FUNCTION "GestStazione_PrioritaSerbatoioPerHMI" : Void
{ S7_Optimized_Access := 'TRUE' }
VERSION : 0.1
   VAR_TEMP
      StazioniConPriorità : Array[0.."K_NumStazione"] of Int;
      StazioniSorgenti : Array[0.."K_NumStazione"] of Int;
      StazioniDestinazioni : Array[0.."K_NumStazione"] of Int;
      CounterStazione : Int;
      OccupazioneArray : Int;
      StazioneDaElenco : Int;
      StazioneVisualizzataHmi : Int;
      LeggiDaPlc : Bool;
      LeggiDaHmi : Bool;
   END_VAR


BEGIN
	REGION Pulizia delle temporanee
	    FOR #CounterStazione := 0 TO "K_NumStazione" DO
	        #StazioniSorgenti[#CounterStazione] :=
	        #StazioniDestinazioni[#CounterStazione] :=
	        #StazioniConPriorità[#CounterStazione] := 0;
	    END_FOR;
	    #StazioneVisualizzataHmi := "PrioritaStazioni".K_StazioneVisualizzata;
	END_REGION ;
	REGION Ricerca stazioni con le priorità
	    #OccupazioneArray := 0;
	    FOR #CounterStazione := 0 TO "K_NumStazione" DO
	        IF "Stazione".S[#CounterStazione].Prm.AbilitazionePriorità.SuEstrazioni OR "Stazione".S[#CounterStazione].Prm.AbilitazionePriorità.SugliArrivi THEN
	            #StazioniConPriorità[#OccupazioneArray] := #CounterStazione;
	            #OccupazioneArray += 1;
	        END_IF;
	    END_FOR;
	END_REGION ;
	REGION Ricerca sorgenti e destinazioni per la stazione visualizzata
	    #OccupazioneArray := 0;
	    FOR #CounterStazione := 0 TO "K_NumStazione" DO
	        IF "Stazione".S[#CounterStazione].Destinazione[#StazioneVisualizzataHmi].IN.Possibile THEN
	            #StazioniSorgenti[#OccupazioneArray] := #CounterStazione;
	            #OccupazioneArray += 1;
	        END_IF;
	    END_FOR;
	    #OccupazioneArray := 0;
	    FOR #CounterStazione := 0 TO "K_NumStazione" DO
	        IF "Stazione".S[#StazioneVisualizzataHmi].Destinazione[#CounterStazione].IN.Possibile THEN
	            #StazioniDestinazioni[#OccupazioneArray] := #CounterStazione;
	            #OccupazioneArray += 1;
	        END_IF;
	    END_FOR;
	END_REGION ;
	REGION Definzione dell'elenco di stazioni da visualizzare ad HMI
	    "PrioritaStazioni".K_StazioniSorgenti := #StazioniSorgenti;
	    "PrioritaStazioni".K_StazioniDestinazioni := #StazioniDestinazioni;
	    "PrioritaStazioni".K_StazioniConPriorità := #StazioniConPriorità;
	END_REGION ;
	REGION Definzione lettura e scrittura
	    #LeggiDaPlc := "PrioritaStazioni".Old_K_StazioneVisualizzata <> "PrioritaStazioni".K_StazioneVisualizzata;

	    #LeggiDaHmi :=  ("PrioritaStazioni".Old_StazioniSorgenti_PrioritàHmi <> "PrioritaStazioni".StazioniSorgenti_PrioritàHmi) OR
	                    ("PrioritaStazioni".Old_StazioniDestinazioni_PrioritàHmi <> "PrioritaStazioni".StazioniDestinazioni_PrioritàHmi);
	    IF #LeggiDaPlc THEN
	        FOR #CounterStazione := 0 TO "K_NumStazione" DO
	            #StazioneDaElenco := #StazioniSorgenti[#CounterStazione];    //Sfoglio l'elenco di stazioni e mi salvo la k
	            "PrioritaStazioni".StazioniSorgenti_PrioritàHmi[#CounterStazione] := "Stazione".S[#StazioneDaElenco].Destinazione[#StazioneVisualizzataHmi].Prm.PrioritaRicezioneProdotto;
	        END_FOR;
	        FOR #CounterStazione := 0 TO "K_NumStazione" DO
	            #StazioneDaElenco := #StazioniDestinazioni[#CounterStazione];    //Sfoglio l'elenco di stazioni e mi salvo la k
	            "PrioritaStazioni".StazioniDestinazioni_PrioritàHmi[#CounterStazione] := "Stazione".S[#StazioneVisualizzataHmi].Destinazione[#StazioneDaElenco].Prm.PrioritaInvioProdotto;
	        END_FOR;
	    END_IF;
	    IF #LeggiDaHmi THEN
	        FOR #CounterStazione := 0 TO "K_NumStazione" DO
	            #StazioneDaElenco := #StazioniSorgenti[#CounterStazione];    //Sfoglio l'elenco di stazioni e mi salvo la k
	            "Stazione".S[#StazioneDaElenco].Destinazione[#StazioneVisualizzataHmi].Prm.PrioritaRicezioneProdotto := "PrioritaStazioni".StazioniSorgenti_PrioritàHmi[#CounterStazione];
	        END_FOR;
	        FOR #CounterStazione := 0 TO "K_NumStazione" DO
	            #StazioneDaElenco := #StazioniDestinazioni[#CounterStazione];    //Sfoglio l'elenco di stazioni e mi salvo la k
	            "Stazione".S[#StazioneVisualizzataHmi].Destinazione[#StazioneDaElenco].Prm.PrioritaInvioProdotto := "PrioritaStazioni".StazioniDestinazioni_PrioritàHmi[#CounterStazione];
	        END_FOR;
	    END_IF;
	    "PrioritaStazioni".Old_StazioniDestinazioni_PrioritàHmi := "PrioritaStazioni".StazioniDestinazioni_PrioritàHmi;
	    "PrioritaStazioni".Old_StazioniSorgenti_PrioritàHmi := "PrioritaStazioni".StazioniSorgenti_PrioritàHmi;
	    "PrioritaStazioni".Old_K_StazioneVisualizzata := "PrioritaStazioni".K_StazioneVisualizzata;
	END_REGION ;

END_FUNCTION

